FUNCTION_BLOCK StartMotorsAndProgramTask EXTENDS TcoAbbRoboticsTask



IF Execute() THEN
	 _blink(inOnTime:=T#500MS,inOffTime:=T#500MS);

  	IF _progress = 0 THEN
		IF NOT __ISVALIDREF(inoControl) THEN
			_varInfo :=__VARINFO(inoControl);
			Messenger.Programming(_sb.Clear().Append('<#Invalid reference: #>').Append(_varInfo.Symbol).ToString()).Pin();
		ELSIF NOT __ISVALIDREF(inoConfig) THEN                                                  
			_varInfo :=__VARINFO(inoConfig);                                                    
			Messenger.Programming(_sb.Clear().Append('<#Invalid reference: #>').Append(_varInfo.Symbol).ToString()).Pin();
		ELSIF NOT __ISVALIDREF(inoStatus) THEN                                                  
			_varInfo :=__VARINFO(inoStatus);                                                    
			Messenger.Programming(_sb.Clear().Append('<#Invalid reference: #>').Append(_varInfo.Symbol).ToString()).Pin();
		ELSE

			_progress := _progress + 1;

		END_IF

	END_IF
	IF _progress = 1 THEN
	
		_varInfo :=__VARINFO( inoStatus.State.AutoOn);                                                
		THIS^.Messenger.OnCondition(_infoTimer.Q AND NOT inoStatus.State.AutoOn).Warning(_sb.Clear().Append('<#Waiting for Auto signal! #>').Append(_varInfo.Symbol).ToString());
		Messenger.Warning('<#Robot is not in Auto#>');
		IF  inoStatus.State.AutoOn THEN
			_progress := _progress + 1;
		END_IF;
	END_IF;
	
	
	IF _progress = 2 THEN	
		Messenger.Debug('<#Robot Error Reset#>');
		inoControl.ResetError := inoStatus.State.Error AND _blink.outQ;
		IF NOT inoStatus.State.Error THEN
			inoControl.ResetError:=FALSE;
			_progress := _progress + 1;
		END_IF
	END_IF;
	
	IF _progress = 3 THEN	
		Messenger.Debug('<#Robot Emergency Stop Reset#>');
		inoControl.ResetEmgStop := inoStatus.State.EmgStop AND _blink.outQ;
		IF NOT inoStatus.State.EmgStop THEN
			inoControl.ResetEmgStop:=FALSE;
			_progress := _progress + 1;
		END_IF
	END_IF;
		
	
	IF _progress = 4 THEN	
		IF inoStatus.State.Error THEN 
			_progress := 1;
		END_IF
		_varInfo :=__VARINFO( inoStatus.State.MotorOnState);                                                
		THIS^.Messenger.OnCondition(_infoTimer.Q AND NOT inoStatus.State.MotorOnState).Warning(_sb.Clear().Append('<# Waiting for signal: #>').Append(_varInfo.Symbol).ToString());
		_varInfo :=__VARINFO( inoStatus.State.CycleOn);                                                
		THIS^.Messenger.OnCondition(_infoTimer.Q AND NOT inoStatus.State.CycleOn).Warning(_sb.Clear().Append('<# Waiting for signal: #>').Append(_varInfo.Symbol).ToString());
		_varInfo :=__VARINFO( inoStatus.State.Error);                                                
		THIS^.Messenger.OnCondition(_infoTimer.Q AND NOT inoStatus.State.Error).Warning(_sb.Clear().Append('<# Waiting for signal: #>').Append(_varInfo.Symbol).ToString());
	
		inoControl.MotorOnAndStart:=_blink.outQ;	
		IF inoStatus.State.MotorOnState AND inoStatus.State.CycleOn AND NOT inoStatus.State.Error THEN
			 inoControl.MotorOnAndStart:=FALSE;
			_progress := _progress + 1;
		END_IF
	END_IF;		
	
	
	
	
    DoneWhen(inoStatus.State.CycleOn AND inoStatus.State.MotorOnState AND NOT inoStatus.State.Error);
    CallTimers(TRUE);
	
	THIS^.ThrowWhen(_errorTimer.Q );
	
END_IF

IF  THIS^.Error AND NOT _errorMessage.Pinned THEN
	THIS^.Restore();
END_IF

METHOD PUBLIC FB_init : BOOL
VAR_INPUT
    bInitRetains : BOOL; // if TRUE, the retain variables are initialized (warm start / cold start)
    bInCopyCode : BOOL; // if TRUE, the instance afterwards gets moved into the copy code (online change)
    ParentObject : ITcoObject;	
END_VAR
END_METHOD

(*~
	<docu>
		<summary>
			Executes when task is aborted.
		</summary>			
	</docu>	
~*)
METHOD PROTECTED OnAbort
IF  __ISVALIDREF(inoStatus) THEN   THIS^.inoStatus.ActionDescription := '<#Start motors and program was aborted.#>'; END_IF;
END_METHOD

(*~
	<docu>
		<summary>
			Executes when task reaches the ```Done``` state .
		</summary>			
	</docu>	
~*)
METHOD PROTECTED OnDone
IF  __ISVALIDREF(inoStatus) THEN   THIS^.inoStatus.ActionDescription := '<#Start motors and program finished successfully.#>'; END_IF;
_progress:=0;
END_METHOD

METHOD PROTECTED OnError

VAR
	description: STRING;
END_VAR
description := '<#Start motors and program finished with error.#>'; 
IF  __ISVALIDREF(inoStatus) THEN   THIS^.inoStatus.ActionDescription := description; END_IF;
THIS^._errorMessage.Error(_sb.Clear().Append(description).Append(' To restore acknowledge this alarm.').ToString()).Pin();
END_METHOD

METHOD PROTECTED OnStart
IF  __ISVALIDREF(inoStatus) THEN  THIS^.inoStatus.ActionDescription := '<#Start motors and program started.#>'; END_IF; 
CallTimers(FALSE);
END_METHOD

(*~
	<docu>
		<summary>
			Restores this instance to the Ready state. Can be called explicitly or from within one of the restore mechanisms.
			<para>
				See also <see cref="PlcDocu.TcoCore.TcoTask.AutoRestorable()"/>
			</para>
		</summary>			
	</docu>	
~*)
METHOD Restore : ITcoRestorable
SUPER^.Restore();
END_METHOD

END_FUNCTION_BLOCK

(* stored: Version 1.1.0.1, ProductVersion 3.1.4024.12
   POU StartMotorsAndProgramTask: Id {342f1f3f-14e5-0206-1a0e-8d3dc471a65a}, SpecialFunc None
   Method FB_init: Id {4e2a99be-fa2c-098d-228c-698e5da90eda}
   Method OnAbort: Id {966fb29c-336e-028c-28a6-685597792162}
   Method OnDone: Id {abb85b23-1eff-0032-1367-598a510ae7bb}
   Method OnError: Id {c37e298c-792d-0733-0dca-3c466c4fb480}
   Method OnStart: Id {deef449b-964f-0742-165c-7f41dfe257c7}
   Method Restore: Id {91088ca2-14bd-0b7d-12cd-f7151351e16f} *)
